Staubli VAL3: setView.pgx

public program setView(bool x_bLarge (dimensions=1))
begin
  // look if to enlarge the screen
  if x_bLarge
    nTopX[1]=nTopX
    nTopX=0
    nBottomX[1]=nBottomX
    nBottomX=38
  else
    nTopX=nTopX[1]
    nBottomX=nBottomX[1]
  endIf
  bUseRefresh=true
end
